FUNCTION_BLOCK PuestoCupula
VAR_INPUT
	Reset:BOOL;
	SFCreset:BOOL;
	Enable:BOOL;
	FinCiclo:BOOL;
	SensorPallet:BOOL;
	Pulsador1 AT %I*:BOOL;
	NumeroDePuesto :INT;	
	SelectorByPass AT %I*:BOOL;
	Pass AT %I*:BOOL;
	Fail AT %I*:BOOL;
	
	SensorPieza1 AT %I*:BOOL;
	SensorPieza2 AT %I*:BOOL;
	
	SensorCupulaAtras AT%I*:BOOL;
	SensorCupulaAdelante AT%I*:BOOL;
END_VAR
VAR_OUTPUT
	
	Ready AT %Q*:BOOL;
	StopperOFF AT %Q*:BOOL;
	Centrador AT%Q*:BOOL;
	Actuador AT%Q*:BOOL;
	LuzAmbar AT%Q*:BOOL;
	SalidaAlarma:BOOL;
	EnMovimiento:BOOL;
	EsperandoPalet:BOOL;
	RetrasoPuesto :INT;
	FinPuesto:BOOL;
	
	CupulaAdelante AT%Q*:BOOL;
	CupulaAtras AT%Q*:BOOL;

	
	
END_VAR

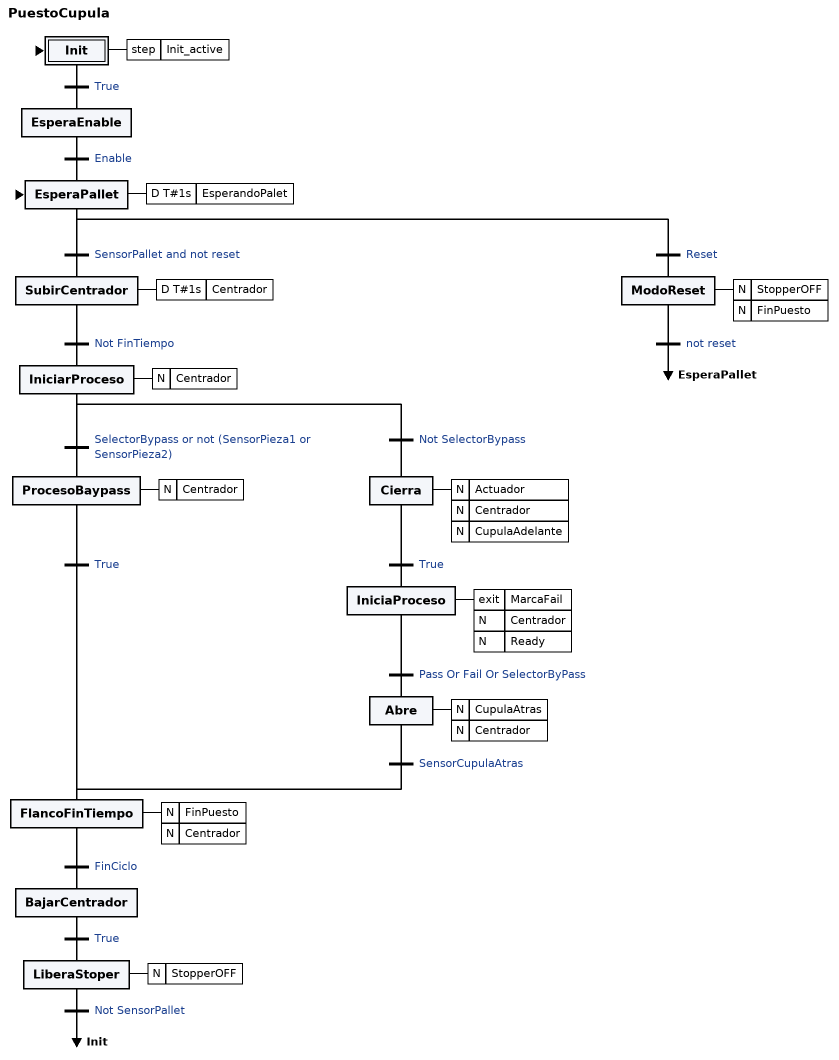
INITIAL_STEP Init:
    Init_active(N);  // step action
END_STEP
TRANSITION FROM Init TO EsperaEnable
    := True;
END_TRANSITION
STEP EsperaEnable:
END_STEP
TRANSITION FROM EsperaEnable TO EsperaPallet
    := Enable;
END_TRANSITION
STEP EsperaPallet:
    EsperandoPalet(D, T#1s);
END_STEP
TRANSITION FROM EsperaPallet TO SubirCentrador
    := SensorPallet and not reset;
END_TRANSITION
STEP SubirCentrador:  // min time T#2s
    Centrador(D, T#1s);
END_STEP
TRANSITION FROM SubirCentrador TO IniciarProceso
    := Not FinTiempo;
END_TRANSITION
STEP IniciarProceso:
    Centrador(N);
END_STEP
TRANSITION FROM IniciarProceso TO ProcesoBaypass
    := SelectorBypass or not (SensorPieza1 or SensorPieza2);
END_TRANSITION
STEP ProcesoBaypass:
    Centrador(N);
END_STEP
TRANSITION FROM ProcesoBaypass TO FlancoFinTiempo
    := True;
END_TRANSITION
TRANSITION FROM IniciarProceso TO Cierra
    := Not SelectorBypass;
END_TRANSITION
STEP Cierra:  // min time T#3s
    Actuador(N);
    Centrador(N);
    CupulaAdelante(N);
END_STEP
TRANSITION FROM Cierra TO IniciaProceso
    := True;
END_TRANSITION
STEP IniciaProceso:  // min time T#5s
    MarcaFail(P0);  // exit action
    Centrador(N);
    Ready(N);
END_STEP
TRANSITION FROM IniciaProceso TO Abre
    := Pass Or Fail Or SelectorByPass;
END_TRANSITION
STEP Abre:
    CupulaAtras(N);
    Centrador(N);
END_STEP
TRANSITION FROM Abre TO FlancoFinTiempo
    := SensorCupulaAtras;
END_TRANSITION
STEP FlancoFinTiempo:
    FinPuesto(N);
    Centrador(N);
END_STEP
TRANSITION FROM FlancoFinTiempo TO BajarCentrador
    := FinCiclo;
END_TRANSITION
STEP BajarCentrador:  // min time T#1s
END_STEP
TRANSITION FROM BajarCentrador TO LiberaStoper
    := True;
END_TRANSITION
TRANSITION FROM EsperaPallet TO ModoReset
    := Reset;
END_TRANSITION
STEP ModoReset:
    StopperOFF(N);
    FinPuesto(N);
END_STEP
TRANSITION FROM ModoReset TO EsperaPallet
    := not reset;
END_TRANSITION
STEP LiberaStoper:  // min time T#1s
    StopperOFF(N);
END_STEP
TRANSITION FROM LiberaStoper TO Init
    := Not SensorPallet;
END_TRANSITION

ACTION EsperaEnable_active:

END_ACTION

ACTION Init_active:
FinPUesto :=FALSE;
SFCreset:=FALSE;
END_ACTION

ACTION MarcaFail:
IF  Fail = TRUE THEN 
	gvl.FalloPallet[NumeroDePuesto] := TRUE;
END_IF
END_ACTION

END_FUNCTION_BLOCK

(* stored: Version 1.1.0.1, ProductVersion 3.1.4024.12
   POU PuestoCupula: Id {d132c2f5-cd59-48fc-a5f1-6f8931e79e9d}, SpecialFunc None
   Action EsperaEnable_active: Id {9aee0fb4-f6c7-4a0c-9a1d-64dce781193b}
   Action Init_active: Id {207f0eb6-c0fb-4ebe-84ee-758a7add2388}
   Action MarcaFail: Id {3ee8ef46-9afc-47d8-a7f1-b90e8bd584c8} *)
